FUNCTION_BLOCK FB_TelescopeIdleState EXTENDS FB_TelescopeState
VAR_INPUT
END_VAR
VAR_OUTPUT
END_VAR
VAR
END_VAR

//
// commands
// 

IF bPark THEN
	pMachine^.State := E_TelescopeState.parking;
	bPark := FALSE;
END_IF

IF bSlew THEN
	pMachine^.State := E_TelescopeState.slewing;
	bSlew := FALSE;
END_IF

IF bTrack THEN
	pMachine^.State := E_TelescopeState.tracking;
	bTrack := FALSE;
END_IF

END_FUNCTION_BLOCK

(* stored: Version 1.1.0.1, ProductVersion 3.1.4024.15
   POU FB_TelescopeIdleState: Id {97cb9578-1d5b-4b37-b757-b2f2bee04a18}, SpecialFunc None *)
